(* Logix 5000 project; controller ProjectTemplate vendor 1 type 14 code 92 rev 34.11; software revision 34.01 *)

MODULES
   Local : vendor 1 type 14 code 92 (ICP 0, rev 34.11)
END_MODULES
